Yaskawa INFORM job: R1_W14,16(0,0)OK-KM.JBI

/JOB
//NAME R1_W14,16(0,0)OK-KM
///FOLDERNAME SCIANA-NOWY-R2-KM
//POS
///NPOS 93,93,0,5,0,0
///TOOL 0
///POSTYPE PULSE
///PULSE
C00000=-76719,27067,-12703,-1851,75531,82265
C00001=-221845,11528,-10687,-35843,76459,22511
C00002=-223898,15400,-5399,-35399,74583,22281
C00003=-224696,17014,-3202,-35233,73827,22198
C00004=-224925,19717,-688,-35188,73602,22179
C00005=-224696,17014,-3202,-35233,73827,22198
C00006=-225261,17174,-2343,-35131,73231,22157
C00007=-225261,17198,-716,-35294,72415,22427
C00008=-225261,17174,-2343,-35131,73231,22157
C00009=-225679,16921,-2293,-35027,72929,22082
C00010=-226650,16415,-2761,-34720,72562,21794
C00011=-225679,16921,-2293,-35027,72929,22082
C00012=-224889,15264,-4529,-35187,73682,22165
C00013=-222855,11289,-9907,-35620,75552,22394
C00014=-219447,-10472,-24872,-64988,60407,26017
C00015=-221941,-5939,-21577,-64020,58945,25442
C00016=-222901,-4078,-20190,-63638,58379,25222
C00017=-223193,-1318,-17925,-63523,58205,25156
C00018=-222901,-4078,-20190,-63638,58379,25222
C00019=-223623,-4073,-20322,-63340,57962,25050
C00020=-224839,-4705,-20836,-62913,57187,24828
C00021=-223623,-4073,-20322,-63340,57962,25050
C00022=-223171,-4056,-22765,-62690,58966,24418
C00023=-223171,-4022,-23364,-62488,59152,24236
C00024=-223131,-4482,-21858,-63116,58620,24792
C00025=-222170,-6353,-23251,-63510,59178,25014
C00026=-219676,-10918,-26561,-64509,60623,25596
C00027=-225804,-33308,-47516,-14649,60735,-3292
C00028=-229095,35993,-508,28233,85172,-10845
C00029=-227688,39932,5922,27900,83007,-10856
C00030=-226790,44519,11564,27698,81729,-10833
C00031=-226790,44416,12047,27716,81416,-10908
C00032=-226790,44519,11564,27698,81729,-10833
C00033=-223138,34268,11,21106,77778,-4533
C00034=-223360,36838,2632,21207,77555,-4651
C00035=-224939,37906,4280,23747,79251,-7336
C00036=-226779,30426,503,28956,74617,-10458
C00037=-225636,31064,1135,28546,74179,-10133
C00038=-226600,30523,599,28893,74548,-10406
C00039=-227148,28589,-2110,29014,75323,-10415
C00040=-228569,23918,-8642,29355,77221,-10462
C00041=-231897,-24783,-37516,60687,63086,-20519
C00042=-228563,-73279,-56420,81123,39929,-27461
C00043=-227220,-4749,6526,101907,37254,-32579
C00044=-224697,6160,12781,100075,35173,-31453
C00045=-224429,9123,15435,100292,34996,-31562
C00046=-224605,11077,17175,100348,35132,-31600
C00047=-230490,15170,11894,82498,48890,-27386
C00048=-229403,17959,22836,97601,46867,-30602
C00049=-228177,18916,23722,97753,46281,-30669
C00050=-229934,17291,15365,83972,48224,-27961
C00051=-229952,16460,11390,81585,48668,-26763
C00052=-229952,16870,13154,82351,48519,-27288
C00053=-230676,14786,11627,82547,49019,-27419
C00054=-237195,-19974,-11699,85770,53273,-29838
C00055=-225804,-33308,-47516,-14649,60735,-18499
C00056=-216281,-27557,-47976,-70560,56032,67196
C00057=-233612,-41384,-47873,-87255,19441,69611
C00058=-238770,-25609,-37442,-79527,16002,66293
C00059=-224737,-6433,-29133,-67659,50241,66287
C00060=-224658,-4960,-27948,-67672,50304,66285
C00061=-239501,-14573,4250,-139591,22189,88446
C00062=-235839,-26774,-7842,-132646,23314,85317
C00063=-221446,-7401,-7934,-79897,48338,74515
C00064=-221541,-8858,-15844,-97554,47314,75397
C00065=-224486,-6509,-14853,-96942,45126,75140
C00066=-224882,-57336,-62686,-67250,43175,22585
C00067=-224791,-6483,-15177,-96721,44888,75014
C00068=-224711,-5022,-14002,-96694,44943,74994
C00069=-224897,-46825,-23767,-88777,38645,34750
C00070=-223107,-56571,-29714,-90277,39873,35762
C00071=-221421,-7980,-10217,-78935,48593,73857
C00072=-222068,-39210,-35412,-13702,43601,27753
C00073=-237445,-29301,-40252,55523,45241,-52581
C00074=-227181,-12576,-1738,104260,26625,-66418
C00075=-225790,-2897,3519,100755,26343,-64671
C00076=-224794,2670,7736,100469,25587,-64507
C00077=-227345,4066,-20439,45016,43012,-47031
C00078=-227097,2962,-21381,44821,42900,-46941
C00079=-224815,34024,73198,137832,37092,-83752
C00080=-224835,23817,55025,118968,28678,-72710
C00081=-226919,22764,62484,135058,37527,-82603
C00082=-229748,-408,-2265,59693,35840,-55378
C00083=-229756,-2454,-20610,49339,41999,-49414
C00084=-230430,-3870,-11743,81980,33342,-60137
C00085=-228081,476,-9013,80437,31765,-59410
C00086=-227095,2175,-8898,78795,31235,-58593
C00087=-228071,1861,-8194,80097,31801,-59232
C00088=-227824,748,-9130,80012,31625,-59198
C00089=-227182,19166,41060,115201,33274,-77620
C00090=-230210,6740,30504,113250,35213,-76901
C00091=-237374,-72574,-67689,58599,66595,-55096
C00092=-143354,-69704,-89188,36188,66672,-67535
BC00000=238873,825705,1030015
BC00001=395849,1115251,786663
BC00002=395849,1115251,786663
BC00003=395849,1115251,786663
BC00004=395849,1115251,786663
BC00005=395849,1115251,786663
BC00006=395849,1115251,786663
BC00007=395849,1115251,786663
BC00008=395849,1115251,786663
BC00009=395849,1115251,786663
BC00010=395849,1115251,786663
BC00011=395849,1115251,786663
BC00012=395849,1115251,786663
BC00013=395849,1115251,786663
BC00014=395849,1129442,1034997
BC00015=395849,1129442,1034997
BC00016=395849,1129442,1034997
BC00017=395849,1129442,1034997
BC00018=395849,1129442,1034997
BC00019=395849,1129442,1034997
BC00020=395849,1129442,1034997
BC00021=395849,1129442,1034997
BC00022=395849,1129442,1024244
BC00023=395849,1129442,1024244
BC00024=395849,1129442,1034997
BC00025=395849,1129442,1034997
BC00026=395849,1129442,1034997
BC00027=395849,1132825,1071944
BC00028=395849,1106481,732774
BC00029=395849,1106481,732774
BC00030=395849,1106481,732774
BC00031=395849,1106481,732774
BC00032=395849,1106481,732774
BC00033=395849,1106481,732774
BC00034=395849,1106481,732774
BC00035=395849,1106481,732774
BC00036=395849,1106481,732774
BC00037=395849,1106481,732774
BC00038=395849,1106481,732774
BC00039=395849,1106481,732774
BC00040=395849,1106481,732774
BC00041=395849,1094194,865071
BC00042=395849,1092013,958243
BC00043=395849,1089311,1073599
BC00044=395849,1089311,1073599
BC00045=395849,1089311,1073599
BC00046=395849,1089311,1073599
BC00047=395849,1089311,1073599
BC00048=395849,1089311,1073599
BC00049=395849,1089311,1073599
BC00050=395849,1089311,1073599
BC00051=395849,1089311,1073599
BC00052=395849,1089311,1073599
BC00053=395849,1089311,1073599
BC00054=395849,1089311,1073599
BC00055=392999,1121081,1071944
BC00056=395849,1133137,679894
BC00057=395848,1133137,679891
BC00058=395848,1133137,679891
BC00059=395849,1133137,679894
BC00060=395849,1133137,679894
BC00061=395848,1133137,679891
BC00062=395848,1133137,679891
BC00063=395849,1133137,679894
BC00064=395849,1133315,941889
BC00065=395849,1133315,941889
BC00066=353955,1125272,938514
BC00067=395849,1133315,941889
BC00068=395849,1133315,941889
BC00069=353465,1125178,938475
BC00070=353465,1125178,938475
BC00071=395849,1133315,941889
BC00072=395849,1122141,904437
BC00073=395849,1101764,864956
BC00074=395848,1101762,864954
BC00075=395848,1101762,864954
BC00076=395848,1101762,864954
BC00077=395849,1101764,864956
BC00078=395849,1101764,864956
BC00079=395848,1101762,864954
BC00080=395848,1101762,864954
BC00081=395848,1101762,864954
BC00082=395849,1101764,864956
BC00083=395849,1101764,864956
BC00084=395849,1100794,989313
BC00085=395849,1100794,989313
BC00086=395849,1100793,989310
BC00087=395849,1100794,989313
BC00088=395849,1100794,989313
BC00089=395849,1100794,989313
BC00090=395849,1100794,989313
BC00091=395849,1100794,989313
BC00092=361025,706112,1026895
///POSTYPE BASE
///RECTAN
///RCONF 0,0,0,0,0,0,0,0,0,0,0,0,0,0,0,0,0,0,0,0,0,0,0,0
P00006=0.222,-3.123,-1.508,0.0000,0.0000,0.0000
P00021=-0.225,-6.128,-0.405,0.0000,0.0000,0.0000
P00022=0.222,-3.123,-1.508,0.0000,0.0000,0.0000
P00023=0.143,-0.036,0.682,0.0000,0.0000,0.0000
P00024=0.145,-0.552,1.326,0.0000,0.0000,0.0000
//INST
///DATE 2024/07/29 14:00
///ATTR SC,RW
///GROUP1 RB1,BS1
NOP
'r1_W14,16(0,0)
'Path S915
SFTOF
MOVJ C00000 BC00000 VJ=100.00
MOVL C00001 BC00001 V=333.3
MOVL C00002 BC00002 V=250.0
MOVL C00003 BC00003 V=60.0
REFP 3 C00004 BC00004
CALL JOB:SEARCH-R1
SET P021 P006
SFTON P021
MOVL C00005 BC00005 V=60.0
MOVL C00006 BC00006 V=60.0
REFP 3 C00007 BC00007
CALL JOB:SEARCH-R1
SET P021 P006
SFTON P021
MOVL C00008 BC00008 V=60.0
MOVL C00009 BC00009 V=60.0
REFP 3 C00010 BC00010
CALL JOB:SEARCH-R1
SET P021 P006
SFTON P021
MOVL C00011 BC00011 V=60.0
MOVL C00012 BC00012 V=166.7
MOVL C00013 BC00013 V=166.7
'Path S795 (for W413)
SFTOF
MOVL C00014 BC00014 V=166.7
MOVL C00015 BC00015 V=166.7
MOVL C00016 BC00016 V=60.0
REFP 3 C00017 BC00017
CALL JOB:SEARCH-R1
SET P022 P006
SFTON P022
MOVL C00018 BC00018 V=60.0
MOVL C00019 BC00019 V=60.0
REFP 3 C00020 BC00020
CALL JOB:SEARCH-R1
SET P022 P006
SFTON P022
MOVL C00021 BC00021 V=60.0
MOVL C00022 BC00022 V=60.0
REFP 3 C00023 BC00023
CALL JOB:SEARCH-R1
SET P022 P006
SFTON P022
MOVL C00024 BC00024 V=166.7
MOVL C00025 BC00025 V=166.7
MOVL C00026 BC00026 V=166.7
MOVJ C00027 BC00027 VJ=100.00
'Path S806 (for W414)
SFTOF
MOVL C00028 BC00028 V=333.3
MOVL C00029 BC00029 V=250.0
MOVL C00030 BC00030 V=60.0
REFP 3 C00031 BC00031
CALL JOB:SEARCH-R1
SET P023 P006
SFTON P023
MOVL C00032 BC00032 V=60.0
MOVL C00033 BC00033 V=60.0
REFP 3 C00034 BC00034
CALL JOB:SEARCH-R1
SET P023 P006
SFTON P023
MOVL C00035 BC00035 V=60.0
MOVL C00036 BC00036 V=60.0
REFP 3 C00037 BC00037
CALL JOB:SEARCH-R1
SET P023 P006
SFTON P023
MOVL C00038 BC00038 V=60.0
MOVL C00039 BC00039 V=166.7
MOVL C00040 BC00040 V=166.7
MOVJ C00041 BC00041 VJ=100.00
'Path VIA1130
SFTOF
MOVJ C00042 BC00042 VJ=100.00
'Path S807 (for W414)
SFTOF
MOVJ C00043 BC00043 VJ=100.00
MOVJ C00044 BC00044 VJ=100.00
MOVL C00045 BC00045 V=60.0
REFP 3 C00046 BC00046
CALL JOB:SEARCH-R1
SET P024 P006
SFTON P024
COMM MOVL C00047 BC00047 V=60.0
MOVL C00048 BC00048 V=60.0
REFP 3 C00049 BC00049
CALL JOB:SEARCH-R1
SET P024 P006
SFTON P024
MOVL C00050 BC00050 V=60.0
REFP 3 C00051 BC00051
CALL JOB:SEARCH-R1
SET P024 P006
SFTON P024
MOVL C00052 BC00052 V=116.7
MOVL C00053 BC00053 V=333.3
MOVL C00054 BC00054 V=333.3
MOVJ C00055 BC00055 VJ=100.00
'Path W1128
SFTOF
SFTON P022
MOVJ C00056 BC00056 VJ=100.00
MOVJ C00057 BC00057 VJ=100.00
MOVL C00058 BC00058 V=100.0 PL=0
REFP 1 C00059 BC00059
REFP 2 C00060 BC00060
MACRO1 MJ#(0) ARGF7
ARCON
SFTON P021
MOVL C00061 BC00061 V=12.5
ARCOF
MOVL C00062 BC00062 V=166.7
MOVL C00063 BC00063 V=166.7
SFTOF
'Path W1129
SFTOF
SFTON P022
MOVJ C00064 BC00064 VJ=100.00
MOVJ C00065 BC00065 VJ=100.00
MOVL C00066 BC00066 V=166.7 PL=0
REFP 1 C00067 BC00067
REFP 2 C00068 BC00068
MACRO1 MJ#(0) ARGF7
ARCON
SFTON P021
MOVL C00069 BC00069 V=12.5
ARCOF
MOVL C00070 BC00070 V=166.7
MOVL C00071 BC00071 V=166.7
SFTOF
'Path VIA1131
SFTOF
MOVJ C00072 BC00072 VJ=100.00
'Path W868
SFTOF
SFTON P024
MOVJ C00073 BC00073 VJ=100.00
MOVJ C00074 BC00074 VJ=45.00
MOVJ C00075 BC00075 VJ=100.00
MOVL C00076 BC00076 V=100.0 PL=0
REFP 1 C00077 BC00077
REFP 2 C00078 BC00078
MACRO1 MJ#(0) ARGF10
ARCON
SFTON P023
MOVL C00079 BC00079 V=8.3
MOVL C00080 BC00080 V=8.3
ARCOF
MOVL C00081 BC00081 V=166.7
MOVL C00082 BC00082 V=166.7
MOVL C00083 BC00083 V=166.7
SFTOF
'Path W1127
SFTOF
'Path W1126
SFTOF
SFTON P024
MOVJ C00084 BC00084 VJ=100.00
MOVJ C00085 BC00085 VJ=100.00
MOVL C00086 BC00086 V=100.0 PL=0
REFP 1 C00087 BC00087
REFP 2 C00088 BC00088
MACRO1 MJ#(0) ARGF10
ARCON
SFTON P023
MOVL C00089 BC00089 V=8.3
ARCOF
MOVL C00090 BC00090 V=166.7
MOVL C00091 BC00091 V=333.3
MOVJ C00092 BC00092 VJ=100.00
SFTOF
END
